// TIA Portal V16 export
// export: Created 2021-09-03T12:34:40.7779124Z, ExportSetting WithDefaults, DisplayName Totally Integrated Automation Portal, DisplayVersion V16 Update 3, DisplayName TIA Portal Version Control Interface, DisplayVersion V16 Update 2, DisplayName TIA Portal Openness, DisplayVersion V16 Update 3, DisplayName TIA Portal Teamcenter Gateway, DisplayVersion V16, DisplayName STEP 7 Professional, DisplayVersion V16 Update 3, DisplayName STEP 7 Safety, DisplayVersion V16, DisplayName WinCC Advanced, DisplayVersion V16 Update 3
DATA_BLOCK "dtUfSeq"   // DB16
{ S7_Optimized_Access := 'FALSE' }
VERSION : 0.1
// stored: AutoNumber true, DBAccessibleFromOPCUA true, IsOnlyStoredInLoadMemory false, IsWriteProtectedInAS false
   VAR RETAIN
      START : "Sequence";
      STOP : "Sequence";
      HW : "Sequence";
      HW_A : "Sequence";
      CEB1 : "Sequence";
      CEB1_A : "Sequence";
      CEB2 : "Sequence";
      CEB2_A : "Sequence";
   END_VAR
BEGIN
   START.devOn[1,6] := 1;
   START.devOn[2,1] := 1;
   START.devOn[2,6] := 1;
   START.delay[1..2] := 5;
   STOP.devOn[1,1] := 1;
   STOP.devOn[1,6] := 1;
   STOP.devOn[2,6] := 1;
   STOP.delay[1..2] := 5;
   STOP.delay[3] := 1;
   HW.devOn[1,7] := 1;
   HW.devOn[2,2] := 1;
   HW.devOn[2,7] := 1;
   HW.devOn[3,2..3] := 1;
   HW.devOn[3,7] := 1;
   HW.devOn[4,2..3] := 1;
   HW.devOn[4,5] := 1;
   HW.devOn[4,7] := 1;
   HW.devOn[5,2..3] := 1;
   HW.devOn[5,7] := 1;
   HW.devOn[6,2] := 1;
   HW.devOn[6,7] := 1;
   HW.devOn[7,7] := 1;
   HW.devOn[8,7] := 1;
   HW.devOn[8,10] := 1;
   HW.devOn[9,7] := 1;
   HW.devOn[10,7] := 1;
   HW.devOn[10,9] := 1;
   HW.devOn[11,7] := 1;
   HW.devOn[12,1] := 1;
   HW.devOn[12,7] := 1;
   HW.devOn[13,7] := 1;
   HW.delay[1..3] := 5;
   HW.delay[4] := 10;
   HW.delay[5..7] := 5;
   HW.delay[8] := 10;
   HW.delay[9] := 5;
   HW.delay[10] := 10;
   HW.delay[11] := 5;
   HW.delay[12] := 10;
   HW.delay[13] := 5;
   HW.delay[14] := 1;
   HW_A.devOn[1,7] := 1;
   HW_A.devOn[2,2] := 1;
   HW_A.devOn[2,7] := 1;
   HW_A.devOn[3,2] := 1;
   HW_A.devOn[3,4] := 1;
   HW_A.devOn[3,7] := 1;
   HW_A.devOn[4,2] := 1;
   HW_A.devOn[4,4] := 1;
   HW_A.devOn[4,7] := 1;
   HW_A.devOn[4,11] := 1;
   HW_A.devOn[5,2] := 1;
   HW_A.devOn[5,4] := 1;
   HW_A.devOn[5,7] := 1;
   HW_A.devOn[6,2] := 1;
   HW_A.devOn[6,7] := 1;
   HW_A.devOn[7,7] := 1;
   HW_A.devOn[8,7] := 1;
   HW_A.devOn[8,10] := 1;
   HW_A.devOn[9,7] := 1;
   HW_A.devOn[10,7..8] := 1;
   HW_A.devOn[11,7..9] := 1;
   HW_A.devOn[12,7..8] := 1;
   HW_A.devOn[13,7] := 1;
   HW_A.devOn[14,1] := 1;
   HW_A.devOn[14,7] := 1;
   HW_A.devOn[15,7] := 1;
   HW_A.delay[1..3] := 5;
   HW_A.delay[4] := 10;
   HW_A.delay[5..7] := 5;
   HW_A.delay[8] := 10;
   HW_A.delay[9..10] := 5;
   HW_A.delay[11] := 10;
   HW_A.delay[12..13] := 5;
   HW_A.delay[14] := 10;
   HW_A.delay[15] := 5;
   HW_A.delay[16] := 1;
   CEB1.devOn[1,7] := 1;
   CEB1.devOn[2,7..8] := 1;
   CEB1.devOn[3,2] := 1;
   CEB1.devOn[3,7..8] := 1;
   CEB1.devOn[4,2..3] := 1;
   CEB1.devOn[4,7..8] := 1;
   CEB1.devOn[5,2..3] := 1;
   CEB1.devOn[5,5] := 1;
   CEB1.devOn[5,7..8] := 1;
   CEB1.devOn[5,13] := 1;
   CEB1.devOn[6,2..3] := 1;
   CEB1.devOn[6,5] := 1;
   CEB1.devOn[6,7] := 1;
   CEB1.devOn[6,13] := 1;
   CEB1.devOn[7,2..3] := 1;
   CEB1.devOn[7,7] := 1;
   CEB1.devOn[8,2] := 1;
   CEB1.devOn[8,7] := 1;
   CEB1.devOn[9,7] := 1;
   CEB1.devOn[10,7] := 1;
   CEB1.devOn[10,10] := 1;
   CEB1.devOn[11,7] := 1;
   CEB1.devOn[12,7] := 1;
   CEB1.devOn[12,9] := 1;
   CEB1.devOn[13,7..9] := 1;
   CEB1.devOn[14,7] := 1;
   CEB1.devOn[14,9] := 1;
   CEB1.devOn[15,7] := 1;
   CEB1.devOn[16,2] := 1;
   CEB1.devOn[16,7] := 1;
   CEB1.devOn[17,2..3] := 1;
   CEB1.devOn[17,7] := 1;
   CEB1.devOn[18,2..3] := 1;
   CEB1.devOn[18,5] := 1;
   CEB1.devOn[18,7] := 1;
   CEB1.devOn[19,2..3] := 1;
   CEB1.devOn[19,7] := 1;
   CEB1.devOn[20,2] := 1;
   CEB1.devOn[20,7] := 1;
   CEB1.devOn[21,7] := 1;
   CEB1.devOn[22,7] := 1;
   CEB1.devOn[22,10] := 1;
   CEB1.devOn[23,7] := 1;
   CEB1.devOn[24,7] := 1;
   CEB1.devOn[24,9] := 1;
   CEB1.devOn[25,7..9] := 1;
   CEB1.devOn[26,7] := 1;
   CEB1.devOn[26,9] := 1;
   CEB1.devOn[27,7] := 1;
   CEB1.devOn[28,2] := 1;
   CEB1.devOn[28,7] := 1;
   CEB1.devOn[29,2..3] := 1;
   CEB1.devOn[29,7] := 1;
   CEB1.devOn[30,2..3] := 1;
   CEB1.devOn[30,5] := 1;
   CEB1.devOn[30,7] := 1;
   CEB1.devOn[31,2..3] := 1;
   CEB1.devOn[31,8] := 1;
   CEB1.devOn[32,2] := 1;
   CEB1.devOn[32,7] := 1;
   CEB1.devOn[33,7] := 1;
   CEB1.devOn[34,7] := 1;
   CEB1.devOn[34,10] := 1;
   CEB1.devOn[35,7] := 1;
   CEB1.devOn[36,7] := 1;
   CEB1.devOn[36,9] := 1;
   CEB1.devOn[37,7..9] := 1;
   CEB1.devOn[38,7] := 1;
   CEB1.devOn[38,9] := 1;
   CEB1.devOn[39,7] := 1;
   CEB1.devOn[40,1] := 1;
   CEB1.devOn[40,7] := 1;
   CEB1.devOn[41,7] := 1;
   CEB1.delay[1..4] := 5;
   CEB1.delay[5] := 10;
   CEB1.delay[6..8] := 5;
   CEB1.delay[9..10] := 10;
   CEB1.delay[11..12] := 5;
   CEB1.delay[13] := 10;
   CEB1.delay[14..17] := 5;
   CEB1.delay[18] := 10;
   CEB1.delay[19..21] := 5;
   CEB1.delay[22] := 10;
   CEB1.delay[23..24] := 5;
   CEB1.delay[25] := 10;
   CEB1.delay[26..29] := 5;
   CEB1.delay[30] := 10;
   CEB1.delay[31..33] := 5;
   CEB1.delay[34] := 10;
   CEB1.delay[35..36] := 5;
   CEB1.delay[37] := 10;
   CEB1.delay[38..39] := 5;
   CEB1.delay[40] := 10;
   CEB1.delay[41] := 5;
   CEB1.delay[42] := 1;
   CEB1_A.devOn[1,1..6] := false;
   CEB1_A.devOn[1,7] := 1;
   CEB1_A.devOn[1,8..16] := false;
   CEB1_A.devOn[2,1..6] := false;
   CEB1_A.devOn[2,7..8] := 1;
   CEB1_A.devOn[2,9..16] := false;
   CEB1_A.devOn[3,1] := false;
   CEB1_A.devOn[3,2] := 1;
   CEB1_A.devOn[3,3..6] := false;
   CEB1_A.devOn[3,7..8] := 1;
   CEB1_A.devOn[3,9..16] := false;
   CEB1_A.devOn[4,1] := false;
   CEB1_A.devOn[4,2] := 1;
   CEB1_A.devOn[4,4] := 1;
   CEB1_A.devOn[4,5..6] := false;
   CEB1_A.devOn[4,7..8] := 1;
   CEB1_A.devOn[4,9..16] := false;
   CEB1_A.devOn[5,1] := false;
   CEB1_A.devOn[5,2] := 1;
   CEB1_A.devOn[5,4] := 1;
   CEB1_A.devOn[5,6] := false;
   CEB1_A.devOn[5,7..8] := 1;
   CEB1_A.devOn[5,9..10] := false;
   CEB1_A.devOn[5,11] := 1;
   CEB1_A.devOn[5,12] := false;
   CEB1_A.devOn[5,13] := 1;
   CEB1_A.devOn[5,14..16] := false;
   CEB1_A.devOn[6,1] := false;
   CEB1_A.devOn[6,2] := 1;
   CEB1_A.devOn[6,4] := 1;
   CEB1_A.devOn[6,6] := false;
   CEB1_A.devOn[6,7] := 1;
   CEB1_A.devOn[6,8..10] := false;
   CEB1_A.devOn[6,11] := 1;
   CEB1_A.devOn[6,12] := false;
   CEB1_A.devOn[6,13] := 1;
   CEB1_A.devOn[6,14..16] := false;
   CEB1_A.devOn[7,1] := false;
   CEB1_A.devOn[7,2] := 1;
   CEB1_A.devOn[7,4] := 1;
   CEB1_A.devOn[7,5..6] := false;
   CEB1_A.devOn[7,7] := 1;
   CEB1_A.devOn[7,8..16] := false;
   CEB1_A.devOn[8,1] := false;
   CEB1_A.devOn[8,2] := 1;
   CEB1_A.devOn[8,3..6] := false;
   CEB1_A.devOn[8,7] := 1;
   CEB1_A.devOn[8,8..16] := false;
   CEB1_A.devOn[9,1..6] := false;
   CEB1_A.devOn[9,7] := 1;
   CEB1_A.devOn[9,8..16] := false;
   CEB1_A.devOn[10,1..6] := false;
   CEB1_A.devOn[10,7] := 1;
   CEB1_A.devOn[10,8..9] := false;
   CEB1_A.devOn[10,10] := 1;
   CEB1_A.devOn[10,11..16] := false;
   CEB1_A.devOn[11,1..6] := false;
   CEB1_A.devOn[11,7] := 1;
   CEB1_A.devOn[11,8..16] := false;
   CEB1_A.devOn[12,1..6] := false;
   CEB1_A.devOn[12,7] := 1;
   CEB1_A.devOn[12,8] := false;
   CEB1_A.devOn[12,9] := 1;
   CEB1_A.devOn[12,10..16] := false;
   CEB1_A.devOn[13,1..6] := false;
   CEB1_A.devOn[13,7..9] := 1;
   CEB1_A.devOn[13,10..16] := false;
   CEB1_A.devOn[14,1..6] := false;
   CEB1_A.devOn[14,7] := 1;
   CEB1_A.devOn[14,8] := false;
   CEB1_A.devOn[14,9] := 1;
   CEB1_A.devOn[14,10..16] := false;
   CEB1_A.devOn[15,1..6] := false;
   CEB1_A.devOn[15,7] := 1;
   CEB1_A.devOn[15,8..16] := false;
   CEB1_A.devOn[16,1] := false;
   CEB1_A.devOn[16,2] := 1;
   CEB1_A.devOn[16,3..6] := false;
   CEB1_A.devOn[16,7] := 1;
   CEB1_A.devOn[16,8..16] := false;
   CEB1_A.devOn[17,1] := false;
   CEB1_A.devOn[17,2] := 1;
   CEB1_A.devOn[17,4] := 1;
   CEB1_A.devOn[17,5..6] := false;
   CEB1_A.devOn[17,7] := 1;
   CEB1_A.devOn[17,8..16] := false;
   CEB1_A.devOn[18,1] := false;
   CEB1_A.devOn[18,2] := 1;
   CEB1_A.devOn[18,4] := 1;
   CEB1_A.devOn[18,6] := false;
   CEB1_A.devOn[18,7] := 1;
   CEB1_A.devOn[18,8..10] := false;
   CEB1_A.devOn[18,11] := 1;
   CEB1_A.devOn[18,12..16] := false;
   CEB1_A.devOn[19,1] := false;
   CEB1_A.devOn[19,2] := 1;
   CEB1_A.devOn[19,4] := 1;
   CEB1_A.devOn[19,5..6] := false;
   CEB1_A.devOn[19,7] := 1;
   CEB1_A.devOn[19,8..16] := false;
   CEB1_A.devOn[20,1] := false;
   CEB1_A.devOn[20,2] := 1;
   CEB1_A.devOn[20,3..6] := false;
   CEB1_A.devOn[20,7] := 1;
   CEB1_A.devOn[20,8..16] := false;
   CEB1_A.devOn[21,1..6] := false;
   CEB1_A.devOn[21,7] := 1;
   CEB1_A.devOn[21,8..16] := false;
   CEB1_A.devOn[22,1..6] := false;
   CEB1_A.devOn[22,7] := 1;
   CEB1_A.devOn[22,8..9] := false;
   CEB1_A.devOn[22,10] := 1;
   CEB1_A.devOn[22,11..16] := false;
   CEB1_A.devOn[23,1..6] := false;
   CEB1_A.devOn[23,7] := 1;
   CEB1_A.devOn[23,8..16] := false;
   CEB1_A.devOn[24,1..6] := false;
   CEB1_A.devOn[24,7] := 1;
   CEB1_A.devOn[24,8] := false;
   CEB1_A.devOn[24,9] := 1;
   CEB1_A.devOn[24,10..16] := false;
   CEB1_A.devOn[25,1..6] := false;
   CEB1_A.devOn[25,7..9] := 1;
   CEB1_A.devOn[25,10..16] := false;
   CEB1_A.devOn[26,1..6] := false;
   CEB1_A.devOn[26,7] := 1;
   CEB1_A.devOn[26,8] := false;
   CEB1_A.devOn[26,9] := 1;
   CEB1_A.devOn[26,10..16] := false;
   CEB1_A.devOn[27,1..6] := false;
   CEB1_A.devOn[27,7] := 1;
   CEB1_A.devOn[27,8..16] := false;
   CEB1_A.devOn[28,1] := false;
   CEB1_A.devOn[28,2] := 1;
   CEB1_A.devOn[28,3..6] := false;
   CEB1_A.devOn[28,7] := 1;
   CEB1_A.devOn[28,8..16] := false;
   CEB1_A.devOn[29,1] := false;
   CEB1_A.devOn[29,2] := 1;
   CEB1_A.devOn[29,3] := false;
   CEB1_A.devOn[29,4] := 1;
   CEB1_A.devOn[29,5..6] := false;
   CEB1_A.devOn[29,7] := 1;
   CEB1_A.devOn[29,8..16] := false;
   CEB1_A.devOn[30,1] := false;
   CEB1_A.devOn[30,2] := 1;
   CEB1_A.devOn[30,3] := false;
   CEB1_A.devOn[30,4] := 1;
   CEB1_A.devOn[30,5..6] := false;
   CEB1_A.devOn[30,7] := 1;
   CEB1_A.devOn[30,8..10] := false;
   CEB1_A.devOn[30,11] := 1;
   CEB1_A.devOn[30,12..16] := false;
   CEB1_A.devOn[31,1] := false;
   CEB1_A.devOn[31,2] := 1;
   CEB1_A.devOn[31,3] := false;
   CEB1_A.devOn[31,4] := 1;
   CEB1_A.devOn[31,5..6] := false;
   CEB1_A.devOn[31,7] := 1;
   CEB1_A.devOn[31,8..16] := false;
   CEB1_A.devOn[32,1] := false;
   CEB1_A.devOn[32,2] := 1;
   CEB1_A.devOn[32,3..6] := false;
   CEB1_A.devOn[32,7] := 1;
   CEB1_A.devOn[32,8..16] := false;
   CEB1_A.devOn[33,1..6] := false;
   CEB1_A.devOn[33,7] := 1;
   CEB1_A.devOn[33,8..16] := false;
   CEB1_A.devOn[34,1..6] := false;
   CEB1_A.devOn[34,7] := 1;
   CEB1_A.devOn[34,8..9] := false;
   CEB1_A.devOn[34,10] := 1;
   CEB1_A.devOn[34,11..16] := false;
   CEB1_A.devOn[35,1..6] := false;
   CEB1_A.devOn[35,7] := 1;
   CEB1_A.devOn[35,8..16] := false;
   CEB1_A.devOn[36,1..6] := false;
   CEB1_A.devOn[36,7] := 1;
   CEB1_A.devOn[36,8] := false;
   CEB1_A.devOn[36,9] := 1;
   CEB1_A.devOn[36,10..16] := false;
   CEB1_A.devOn[37,1..6] := false;
   CEB1_A.devOn[37,7..9] := 1;
   CEB1_A.devOn[37,10..16] := false;
   CEB1_A.devOn[38,1..6] := false;
   CEB1_A.devOn[38,7] := 1;
   CEB1_A.devOn[38,8] := false;
   CEB1_A.devOn[38,9] := 1;
   CEB1_A.devOn[38,10..16] := false;
   CEB1_A.devOn[39,1..6] := false;
   CEB1_A.devOn[39,7] := 1;
   CEB1_A.devOn[39,8..16] := false;
   CEB1_A.devOn[40,1] := 1;
   CEB1_A.devOn[40,2..6] := false;
   CEB1_A.devOn[40,7] := 1;
   CEB1_A.devOn[40,8..16] := false;
   CEB1_A.devOn[41,1..6] := false;
   CEB1_A.devOn[41,7] := 1;
   CEB1_A.devOn[41,8..16] := false;
   CEB1_A.delay[1..4] := 5;
   CEB1_A.delay[5] := 10;
   CEB1_A.delay[6..8] := 5;
   CEB1_A.delay[9..10] := 10;
   CEB1_A.delay[11..12] := 5;
   CEB1_A.delay[13] := 10;
   CEB1_A.delay[14..17] := 5;
   CEB1_A.delay[18] := 10;
   CEB1_A.delay[19..21] := 5;
   CEB1_A.delay[22] := 10;
   CEB1_A.delay[23..24] := 5;
   CEB1_A.delay[25] := 10;
   CEB1_A.delay[26..29] := 5;
   CEB1_A.delay[30] := 10;
   CEB1_A.delay[31..33] := 5;
   CEB1_A.delay[34] := 10;
   CEB1_A.delay[35..36] := 5;
   CEB1_A.delay[37] := 10;
   CEB1_A.delay[38..39] := 5;
   CEB1_A.delay[40] := 10;
   CEB1_A.delay[41] := 5;
   CEB1_A.delay[42] := 1;
   CEB2.devOn[1,1..6] := false;
   CEB2.devOn[1,7] := 1;
   CEB2.devOn[1,8..16] := false;
   CEB2.devOn[2,1..6] := false;
   CEB2.devOn[2,7..8] := 1;
   CEB2.devOn[2,9..16] := false;
   CEB2.devOn[3,1] := false;
   CEB2.devOn[3,2] := 1;
   CEB2.devOn[3,3..6] := false;
   CEB2.devOn[3,7..8] := 1;
   CEB2.devOn[3,9..16] := false;
   CEB2.devOn[4,1] := false;
   CEB2.devOn[4,2..3] := 1;
   CEB2.devOn[4,4..6] := false;
   CEB2.devOn[4,7..8] := 1;
   CEB2.devOn[4,9..16] := false;
   CEB2.devOn[5,1] := false;
   CEB2.devOn[5,2..3] := 1;
   CEB2.devOn[5,4] := false;
   CEB2.devOn[5,5] := 1;
   CEB2.devOn[5,6] := false;
   CEB2.devOn[5,7..8] := 1;
   CEB2.devOn[5,9..11] := false;
   CEB2.devOn[5,12] := 1;
   CEB2.devOn[5,14..16] := false;
   CEB2.devOn[6,1] := false;
   CEB2.devOn[6,2..3] := 1;
   CEB2.devOn[6,4] := false;
   CEB2.devOn[6,5] := 1;
   CEB2.devOn[6,6] := false;
   CEB2.devOn[6,7] := 1;
   CEB2.devOn[6,8..11] := false;
   CEB2.devOn[6,12] := 1;
   CEB2.devOn[6,14..16] := false;
   CEB2.devOn[7,1] := false;
   CEB2.devOn[7,2..3] := 1;
   CEB2.devOn[7,4..6] := false;
   CEB2.devOn[7,7] := 1;
   CEB2.devOn[7,8..16] := false;
   CEB2.devOn[8,1] := false;
   CEB2.devOn[8,2] := 1;
   CEB2.devOn[8,3..6] := false;
   CEB2.devOn[8,7] := 1;
   CEB2.devOn[8,8..16] := false;
   CEB2.devOn[9,1..6] := false;
   CEB2.devOn[9,7] := 1;
   CEB2.devOn[9,8..16] := false;
   CEB2.devOn[10,1..6] := false;
   CEB2.devOn[10,7] := 1;
   CEB2.devOn[10,8..9] := false;
   CEB2.devOn[10,10] := 1;
   CEB2.devOn[10,11..16] := false;
   CEB2.devOn[11,1..6] := false;
   CEB2.devOn[11,7] := 1;
   CEB2.devOn[11,8..16] := false;
   CEB2.devOn[12,1..6] := false;
   CEB2.devOn[12,7] := 1;
   CEB2.devOn[12,8] := false;
   CEB2.devOn[12,9] := 1;
   CEB2.devOn[12,10..16] := false;
   CEB2.devOn[13,1..6] := false;
   CEB2.devOn[13,7..9] := 1;
   CEB2.devOn[13,10..16] := false;
   CEB2.devOn[14,1..6] := false;
   CEB2.devOn[14,7] := 1;
   CEB2.devOn[14,8] := false;
   CEB2.devOn[14,9] := 1;
   CEB2.devOn[14,10..16] := false;
   CEB2.devOn[15,1..6] := false;
   CEB2.devOn[15,7] := 1;
   CEB2.devOn[15,8..16] := false;
   CEB2.devOn[16,1] := false;
   CEB2.devOn[16,2] := 1;
   CEB2.devOn[16,3..6] := false;
   CEB2.devOn[16,7] := 1;
   CEB2.devOn[16,8..16] := false;
   CEB2.devOn[17,1] := false;
   CEB2.devOn[17,2..3] := 1;
   CEB2.devOn[17,4..6] := false;
   CEB2.devOn[17,7] := 1;
   CEB2.devOn[17,8..16] := false;
   CEB2.devOn[18,1] := false;
   CEB2.devOn[18,2..3] := 1;
   CEB2.devOn[18,4] := false;
   CEB2.devOn[18,5] := 1;
   CEB2.devOn[18,6] := false;
   CEB2.devOn[18,7] := 1;
   CEB2.devOn[18,8..16] := false;
   CEB2.devOn[19,1] := false;
   CEB2.devOn[19,2..3] := 1;
   CEB2.devOn[19,4..6] := false;
   CEB2.devOn[19,7] := 1;
   CEB2.devOn[19,8..16] := false;
   CEB2.devOn[20,1] := false;
   CEB2.devOn[20,2] := 1;
   CEB2.devOn[20,3..6] := false;
   CEB2.devOn[20,7] := 1;
   CEB2.devOn[20,8..16] := false;
   CEB2.devOn[21,1..6] := false;
   CEB2.devOn[21,7] := 1;
   CEB2.devOn[21,8..16] := false;
   CEB2.devOn[22,1..6] := false;
   CEB2.devOn[22,7] := 1;
   CEB2.devOn[22,8..9] := false;
   CEB2.devOn[22,10] := 1;
   CEB2.devOn[22,11..16] := false;
   CEB2.devOn[23,1..6] := false;
   CEB2.devOn[23,7] := 1;
   CEB2.devOn[23,8..16] := false;
   CEB2.devOn[24,1..6] := false;
   CEB2.devOn[24,7] := 1;
   CEB2.devOn[24,8] := false;
   CEB2.devOn[24,9] := 1;
   CEB2.devOn[24,10..16] := false;
   CEB2.devOn[25,1..6] := false;
   CEB2.devOn[25,7..9] := 1;
   CEB2.devOn[25,10..16] := false;
   CEB2.devOn[26,1..6] := false;
   CEB2.devOn[26,7] := 1;
   CEB2.devOn[26,8] := false;
   CEB2.devOn[26,9] := 1;
   CEB2.devOn[26,10..16] := false;
   CEB2.devOn[27,1..6] := false;
   CEB2.devOn[27,7] := 1;
   CEB2.devOn[27,8..16] := false;
   CEB2.devOn[28,1] := false;
   CEB2.devOn[28,2] := 1;
   CEB2.devOn[28,3..6] := false;
   CEB2.devOn[28,7] := 1;
   CEB2.devOn[28,8..16] := false;
   CEB2.devOn[29,1] := false;
   CEB2.devOn[29,2..3] := 1;
   CEB2.devOn[29,4..6] := false;
   CEB2.devOn[29,7] := 1;
   CEB2.devOn[29,8..16] := false;
   CEB2.devOn[30,1] := false;
   CEB2.devOn[30,2..3] := 1;
   CEB2.devOn[30,4] := false;
   CEB2.devOn[30,5] := 1;
   CEB2.devOn[30,6] := false;
   CEB2.devOn[30,7] := 1;
   CEB2.devOn[30,8..16] := false;
   CEB2.devOn[31,1] := false;
   CEB2.devOn[31,2..3] := 1;
   CEB2.devOn[31,4..7] := false;
   CEB2.devOn[31,8] := 1;
   CEB2.devOn[31,9..16] := false;
   CEB2.devOn[32,1] := false;
   CEB2.devOn[32,2] := 1;
   CEB2.devOn[32,3..6] := false;
   CEB2.devOn[32,7] := 1;
   CEB2.devOn[32,8..16] := false;
   CEB2.devOn[33,1..6] := false;
   CEB2.devOn[33,7] := 1;
   CEB2.devOn[33,8..16] := false;
   CEB2.devOn[34,1..6] := false;
   CEB2.devOn[34,7] := 1;
   CEB2.devOn[34,8..9] := false;
   CEB2.devOn[34,10] := 1;
   CEB2.devOn[34,11..16] := false;
   CEB2.devOn[35,1..6] := false;
   CEB2.devOn[35,7] := 1;
   CEB2.devOn[35,8..16] := false;
   CEB2.devOn[36,1..6] := false;
   CEB2.devOn[36,7] := 1;
   CEB2.devOn[36,8] := false;
   CEB2.devOn[36,9] := 1;
   CEB2.devOn[36,10..16] := false;
   CEB2.devOn[37,1..6] := false;
   CEB2.devOn[37,7..9] := 1;
   CEB2.devOn[37,10..16] := false;
   CEB2.devOn[38,1..6] := false;
   CEB2.devOn[38,7] := 1;
   CEB2.devOn[38,8] := false;
   CEB2.devOn[38,9] := 1;
   CEB2.devOn[38,10..16] := false;
   CEB2.devOn[39,1..6] := false;
   CEB2.devOn[39,7] := 1;
   CEB2.devOn[39,8..16] := false;
   CEB2.devOn[40,1] := 1;
   CEB2.devOn[40,2..6] := false;
   CEB2.devOn[40,7] := 1;
   CEB2.devOn[40,8..16] := false;
   CEB2.devOn[41,1..6] := false;
   CEB2.devOn[41,7] := 1;
   CEB2.devOn[41,8..16] := false;
   CEB2.delay[1..4] := 5;
   CEB2.delay[5] := 10;
   CEB2.delay[6..8] := 5;
   CEB2.delay[9..10] := 10;
   CEB2.delay[11..12] := 5;
   CEB2.delay[13] := 10;
   CEB2.delay[14..17] := 5;
   CEB2.delay[18] := 10;
   CEB2.delay[19..21] := 5;
   CEB2.delay[22] := 10;
   CEB2.delay[23..24] := 5;
   CEB2.delay[25] := 10;
   CEB2.delay[26..29] := 5;
   CEB2.delay[30] := 10;
   CEB2.delay[31..33] := 5;
   CEB2.delay[34] := 10;
   CEB2.delay[35..36] := 5;
   CEB2.delay[37] := 10;
   CEB2.delay[38..39] := 5;
   CEB2.delay[40] := 10;
   CEB2.delay[41] := 5;
   CEB2.delay[42] := 1;
   CEB2_A.devOn[1,1..6] := false;
   CEB2_A.devOn[1,7] := 1;
   CEB2_A.devOn[1,8..16] := false;
   CEB2_A.devOn[2,1..6] := false;
   CEB2_A.devOn[2,7..8] := 1;
   CEB2_A.devOn[2,9..16] := false;
   CEB2_A.devOn[3,1] := false;
   CEB2_A.devOn[3,2] := 1;
   CEB2_A.devOn[3,3..6] := false;
   CEB2_A.devOn[3,7..8] := 1;
   CEB2_A.devOn[3,9..16] := false;
   CEB2_A.devOn[4,1] := false;
   CEB2_A.devOn[4,2] := 1;
   CEB2_A.devOn[4,3] := false;
   CEB2_A.devOn[4,4] := 1;
   CEB2_A.devOn[4,5..6] := false;
   CEB2_A.devOn[4,7..8] := 1;
   CEB2_A.devOn[4,9..16] := false;
   CEB2_A.devOn[5,1] := false;
   CEB2_A.devOn[5,2] := 1;
   CEB2_A.devOn[5,3] := false;
   CEB2_A.devOn[5,4] := 1;
   CEB2_A.devOn[5,5..6] := false;
   CEB2_A.devOn[5,7..8] := 1;
   CEB2_A.devOn[5,9..10] := false;
   CEB2_A.devOn[5,11..12] := 1;
   CEB2_A.devOn[5,14..16] := false;
   CEB2_A.devOn[6,1] := false;
   CEB2_A.devOn[6,2] := 1;
   CEB2_A.devOn[6,3] := false;
   CEB2_A.devOn[6,4] := 1;
   CEB2_A.devOn[6,5..6] := false;
   CEB2_A.devOn[6,7] := 1;
   CEB2_A.devOn[6,8..10] := false;
   CEB2_A.devOn[6,11..12] := 1;
   CEB2_A.devOn[6,14..16] := false;
   CEB2_A.devOn[7,1] := false;
   CEB2_A.devOn[7,2] := 1;
   CEB2_A.devOn[7,3] := false;
   CEB2_A.devOn[7,4] := 1;
   CEB2_A.devOn[7,5..6] := false;
   CEB2_A.devOn[7,7] := 1;
   CEB2_A.devOn[7,8..16] := false;
   CEB2_A.devOn[8,1] := false;
   CEB2_A.devOn[8,2] := 1;
   CEB2_A.devOn[8,3..6] := false;
   CEB2_A.devOn[8,7] := 1;
   CEB2_A.devOn[8,8..16] := false;
   CEB2_A.devOn[9,1..6] := false;
   CEB2_A.devOn[9,7] := 1;
   CEB2_A.devOn[9,8..16] := false;
   CEB2_A.devOn[10,1..6] := false;
   CEB2_A.devOn[10,7] := 1;
   CEB2_A.devOn[10,8..9] := false;
   CEB2_A.devOn[10,10] := 1;
   CEB2_A.devOn[10,11..16] := false;
   CEB2_A.devOn[11,1..6] := false;
   CEB2_A.devOn[11,7] := 1;
   CEB2_A.devOn[11,8..16] := false;
   CEB2_A.devOn[12,1..6] := false;
   CEB2_A.devOn[12,7] := 1;
   CEB2_A.devOn[12,8] := false;
   CEB2_A.devOn[12,9] := 1;
   CEB2_A.devOn[12,10..16] := false;
   CEB2_A.devOn[13,1..6] := false;
   CEB2_A.devOn[13,7..9] := 1;
   CEB2_A.devOn[13,10..16] := false;
   CEB2_A.devOn[14,1..6] := false;
   CEB2_A.devOn[14,7] := 1;
   CEB2_A.devOn[14,8] := false;
   CEB2_A.devOn[14,9] := 1;
   CEB2_A.devOn[14,10..16] := false;
   CEB2_A.devOn[15,1..6] := false;
   CEB2_A.devOn[15,7] := 1;
   CEB2_A.devOn[15,8..16] := false;
   CEB2_A.devOn[16,1] := false;
   CEB2_A.devOn[16,2] := 1;
   CEB2_A.devOn[16,3..6] := false;
   CEB2_A.devOn[16,7] := 1;
   CEB2_A.devOn[16,8..16] := false;
   CEB2_A.devOn[17,1] := false;
   CEB2_A.devOn[17,2] := 1;
   CEB2_A.devOn[17,3] := false;
   CEB2_A.devOn[17,4] := 1;
   CEB2_A.devOn[17,5..6] := false;
   CEB2_A.devOn[17,7] := 1;
   CEB2_A.devOn[17,8..16] := false;
   CEB2_A.devOn[18,1] := false;
   CEB2_A.devOn[18,2] := 1;
   CEB2_A.devOn[18,3] := false;
   CEB2_A.devOn[18,4] := 1;
   CEB2_A.devOn[18,5..6] := false;
   CEB2_A.devOn[18,7] := 1;
   CEB2_A.devOn[18,8..10] := false;
   CEB2_A.devOn[18,11] := 1;
   CEB2_A.devOn[18,12..16] := false;
   CEB2_A.devOn[19,1] := false;
   CEB2_A.devOn[19,2] := 1;
   CEB2_A.devOn[19,3] := false;
   CEB2_A.devOn[19,4] := 1;
   CEB2_A.devOn[19,5..6] := false;
   CEB2_A.devOn[19,7] := 1;
   CEB2_A.devOn[19,8..16] := false;
   CEB2_A.devOn[20,1] := false;
   CEB2_A.devOn[20,2] := 1;
   CEB2_A.devOn[20,3..6] := false;
   CEB2_A.devOn[20,7] := 1;
   CEB2_A.devOn[20,8..16] := false;
   CEB2_A.devOn[21,1..6] := false;
   CEB2_A.devOn[21,7] := 1;
   CEB2_A.devOn[21,8..16] := false;
   CEB2_A.devOn[22,1..6] := false;
   CEB2_A.devOn[22,7] := 1;
   CEB2_A.devOn[22,8..9] := false;
   CEB2_A.devOn[22,10] := 1;
   CEB2_A.devOn[22,11..16] := false;
   CEB2_A.devOn[23,1..6] := false;
   CEB2_A.devOn[23,7] := 1;
   CEB2_A.devOn[23,8..16] := false;
   CEB2_A.devOn[24,1..6] := false;
   CEB2_A.devOn[24,7] := 1;
   CEB2_A.devOn[24,8] := false;
   CEB2_A.devOn[24,9] := 1;
   CEB2_A.devOn[24,10..16] := false;
   CEB2_A.devOn[25,1..6] := false;
   CEB2_A.devOn[25,7..9] := 1;
   CEB2_A.devOn[25,10..16] := false;
   CEB2_A.devOn[26,1..6] := false;
   CEB2_A.devOn[26,7] := 1;
   CEB2_A.devOn[26,8] := false;
   CEB2_A.devOn[26,9] := 1;
   CEB2_A.devOn[26,10..16] := false;
   CEB2_A.devOn[27,1..6] := false;
   CEB2_A.devOn[27,7] := 1;
   CEB2_A.devOn[27,8..16] := false;
   CEB2_A.devOn[28,1] := false;
   CEB2_A.devOn[28,2] := 1;
   CEB2_A.devOn[28,3..6] := false;
   CEB2_A.devOn[28,7] := 1;
   CEB2_A.devOn[28,8..16] := false;
   CEB2_A.devOn[29,1] := false;
   CEB2_A.devOn[29,2] := 1;
   CEB2_A.devOn[29,3] := false;
   CEB2_A.devOn[29,4] := 1;
   CEB2_A.devOn[29,5..6] := false;
   CEB2_A.devOn[29,7] := 1;
   CEB2_A.devOn[29,8..16] := false;
   CEB2_A.devOn[30,1] := false;
   CEB2_A.devOn[30,2] := 1;
   CEB2_A.devOn[30,3] := false;
   CEB2_A.devOn[30,4] := 1;
   CEB2_A.devOn[30,5..6] := false;
   CEB2_A.devOn[30,7] := 1;
   CEB2_A.devOn[30,8..10] := false;
   CEB2_A.devOn[30,11] := 1;
   CEB2_A.devOn[30,12..16] := false;
   CEB2_A.devOn[31,1] := false;
   CEB2_A.devOn[31,2] := 1;
   CEB2_A.devOn[31,3] := false;
   CEB2_A.devOn[31,4] := 1;
   CEB2_A.devOn[31,5..6] := false;
   CEB2_A.devOn[31,7] := 1;
   CEB2_A.devOn[31,8..16] := false;
   CEB2_A.devOn[32,1] := false;
   CEB2_A.devOn[32,2] := 1;
   CEB2_A.devOn[32,3..6] := false;
   CEB2_A.devOn[32,7] := 1;
   CEB2_A.devOn[32,8..16] := false;
   CEB2_A.devOn[33,1..6] := false;
   CEB2_A.devOn[33,7] := 1;
   CEB2_A.devOn[33,8..16] := false;
   CEB2_A.devOn[34,1..6] := false;
   CEB2_A.devOn[34,7] := 1;
   CEB2_A.devOn[34,8..9] := false;
   CEB2_A.devOn[34,10] := 1;
   CEB2_A.devOn[34,11..16] := false;
   CEB2_A.devOn[35,1..6] := false;
   CEB2_A.devOn[35,7] := 1;
   CEB2_A.devOn[35,8..16] := false;
   CEB2_A.devOn[36,1..6] := false;
   CEB2_A.devOn[36,7] := 1;
   CEB2_A.devOn[36,8] := false;
   CEB2_A.devOn[36,9] := 1;
   CEB2_A.devOn[36,10..16] := false;
   CEB2_A.devOn[37,1..6] := false;
   CEB2_A.devOn[37,7..9] := 1;
   CEB2_A.devOn[37,10..16] := false;
   CEB2_A.devOn[38,1..6] := false;
   CEB2_A.devOn[38,7] := 1;
   CEB2_A.devOn[38,8] := false;
   CEB2_A.devOn[38,9] := 1;
   CEB2_A.devOn[38,10..16] := false;
   CEB2_A.devOn[39,1..6] := false;
   CEB2_A.devOn[39,7] := 1;
   CEB2_A.devOn[39,8..16] := false;
   CEB2_A.devOn[40,1] := 1;
   CEB2_A.devOn[40,2..6] := false;
   CEB2_A.devOn[40,7] := 1;
   CEB2_A.devOn[40,8..16] := false;
   CEB2_A.devOn[41,1..6] := false;
   CEB2_A.devOn[41,7] := 1;
   CEB2_A.devOn[41,8..16] := false;
   CEB2_A.delay[1..4] := 5;
   CEB2_A.delay[5] := 10;
   CEB2_A.delay[6..8] := 5;
   CEB2_A.delay[9..10] := 10;
   CEB2_A.delay[11..12] := 5;
   CEB2_A.delay[13] := 10;
   CEB2_A.delay[14..17] := 5;
   CEB2_A.delay[18] := 10;
   CEB2_A.delay[19..21] := 5;
   CEB2_A.delay[22] := 10;
   CEB2_A.delay[23..24] := 5;
   CEB2_A.delay[25] := 10;
   CEB2_A.delay[26..29] := 5;
   CEB2_A.delay[30] := 10;
   CEB2_A.delay[31..33] := 5;
   CEB2_A.delay[34] := 10;
   CEB2_A.delay[35..36] := 5;
   CEB2_A.delay[37] := 10;
   CEB2_A.delay[38..39] := 5;
   CEB2_A.delay[40] := 10;
   CEB2_A.delay[41] := 5;
   CEB2_A.delay[42] := 1;
END_DATA_BLOCK
